(* IEC 61131-3 sources: RL_MAR/experiments/comparison/autoplc/results/gpt-4o_20260511_211137/med_87, 1 file *)

(* ---- med_87_1.st ---- *)
FUNCTION_BLOCK WaterDesalination
    VAR_INPUT
        StartButton : BOOL; (* Input for starting the desalination process *)
        StopButton : BOOL; (* Input for stopping the desalination process *)
        SalinitySensor : REAL; (* Input for salinity level measurement *)
    END_VAR

    VAR_OUTPUT
        SeawaterInletValve : BOOL; (* Output for seawater inlet valve control *)
        FreshwaterOutletValve : BOOL; (* Output for freshwater outlet valve control *)
        DesalinationInProgress : BOOL; (* Indicator for an ongoing desalination process *)
    END_VAR

    VAR
        MaxSalinity : REAL := 35.0; (* Maximum allowable salinity in ppm for freshwater *)
        SalinityControlSeconds : INT := 0; (* Timer for salinity control in seconds *)
        TimerTick : BOOL := FALSE; (* Internal flag to simulate timer tick every second *)
    END_VAR

    // Initialization
    MaxSalinity := 35.0;
    SalinityControlSeconds := 0;
    DesalinationInProgress := FALSE;
    SeawaterInletValve := FALSE;
    FreshwaterOutletValve := FALSE;

    // Start/Stop Control
    IF StartButton AND NOT DesalinationInProgress THEN
        DesalinationInProgress := TRUE;
        SeawaterInletValve := TRUE;
        FreshwaterOutletValve := TRUE;
    ELSIF StopButton THEN
        DesalinationInProgress := FALSE;
        SeawaterInletValve := FALSE;
        FreshwaterOutletValve := FALSE;
        SalinityControlSeconds := 0;
    END_IF

    // Simulate a timer tick every second
    IF TimerTick THEN
        SalinityControlSeconds := SalinityControlSeconds + 1;
        TimerTick := FALSE; // Reset the timer tick flag
    END_IF

    // Salinity Monitoring and Control
    IF DesalinationInProgress THEN
        IF SalinityControlSeconds >= 10 THEN
            IF SalinitySensor > MaxSalinity THEN
                FreshwaterOutletValve := FALSE;
            ELSE
                FreshwaterOutletValve := TRUE;
            END_IF
            SalinityControlSeconds := 0; // Reset the timer for the next 10-second interval
        END_IF
    END_IF
END_FUNCTION_BLOCK
